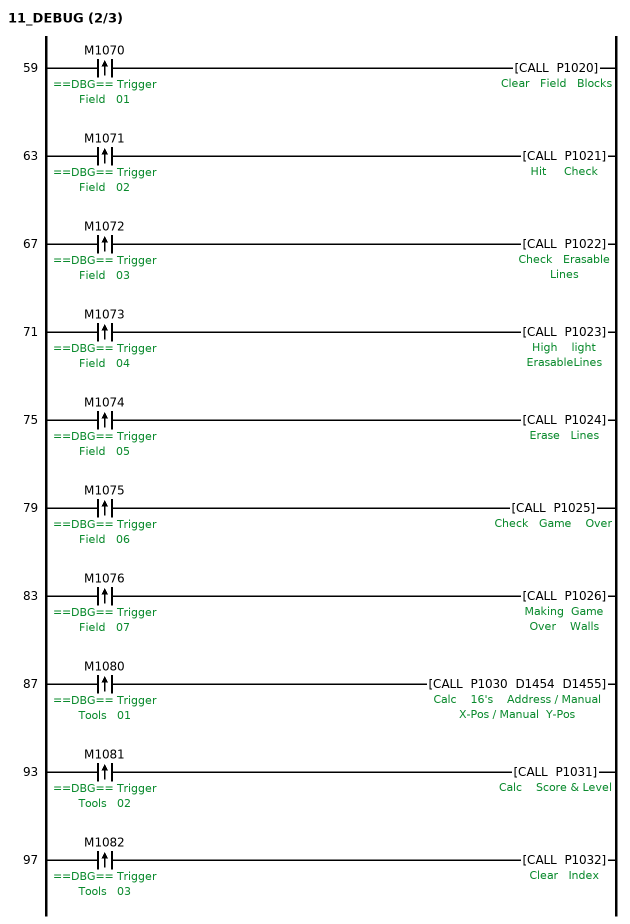
[picture p24: ladder of 11_DEBUG, rungs at steps 59 to 97]
59    LDP     M1070  ; ==DBG== Trigger Field   01
      CALL    P1020  ; Clear   Field   Blocks
63    LDP     M1071  ; ==DBG== Trigger Field   02
      CALL    P1021  ; Hit     Check
67    LDP     M1072  ; ==DBG== Trigger Field   03
      CALL    P1022  ; Check   ErasableLines
71    LDP     M1073  ; ==DBG== Trigger Field   04
      CALL    P1023  ; High    light   ErasableLines
75    LDP     M1074  ; ==DBG== Trigger Field   05
      CALL    P1024  ; Erase   Lines
79    LDP     M1075  ; ==DBG== Trigger Field   06
      CALL    P1025  ; Check   Game    Over
83    LDP     M1076  ; ==DBG== Trigger Field   07
      CALL    P1026  ; Making  Game    Over    Walls
87    LDP     M1080  ; ==DBG== Trigger Tools   01
      CALL    P1030 D1454 D1455  ; Calc    16's    Address / Manual  X-Pos / Manual  Y-Pos
93    LDP     M1081  ; ==DBG== Trigger Tools   02
      CALL    P1031  ; Calc    Score & Level
97    LDP     M1082  ; ==DBG== Trigger Tools   03
      CALL    P1032  ; Clear   Index
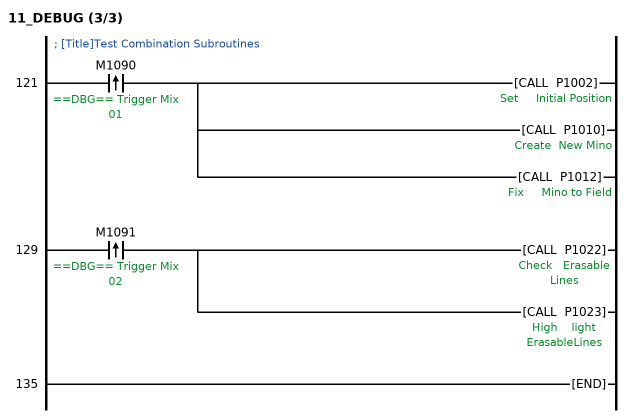
; [Title]Test Combination Subroutines
121   LDP     M1090  ; ==DBG== Trigger Mix     01
      CALL    P1002
      CALL    P1010
      CALL    P1012
129   LDP     M1091  ; ==DBG== Trigger Mix     02
      CALL    P1022
      CALL    P1023
135   END
END_PROGRAM
